TYPE ST_CtrlInRunnerCheck :
STRUCT
	ExternalTrigger			: BOOL; //Optionally start meassurement if the standard trigging is not sufficient 
END_STRUCT
END_TYPE

(* stored: Version 1.1.0.1, ProductVersion 3.1.4024.9
   DUT ST_CtrlInRunnerCheck: Id {5b4e457e-fe41-4ea5-8d9b-162a003a185e} *)
